FUNCTION_BLOCK FB_Alarms
VAR_INPUT
	evEntry			: TcEventEntry;
	bEvt			: BOOL;
	bConfirm		: BOOL;
END_VAR
VAR_OUTPUT
	Q							: BOOL;
END_VAR
VAR
	bInit			: BOOL :=	TRUE;
	rAlarmActivation: Tc2_Standard.R_TRIG;
	rReset			: Tc2_Standard.RS;
END_VAR

IF bInit THEN
	
	SUPER^.CreateEx(evEntry, TRUE, 0);
	bInit := FALSE;

END_IF


IF bEvt  THEN
	SUPER^.Raise (0);
ELSE SUPER^.Clear (0, FALSE);
END_IF


IF bConfirm AND NOT bEvt THEN
	
	SUPER^.Confirm(0);

END_IF


Q := SUPER^.bRaised;

END_FUNCTION_BLOCK

(* stored: Version 1.1.0.1, ProductVersion 3.1.4024.13
   POU FB_Alarms: Id {9692cb57-caf1-482e-b488-a322cd2b915c}, SpecialFunc None *)
